TYPE ST_Base :
STRUCT
    nId : INT;
END_STRUCT
END_TYPE

(* stored: Version 1.1.0.1
   DUT ST_Base: Id {77777777-7777-7777-7777-777777777703} *)
